{attribute 'qualified_only'}
{attribute 'to_string'}
TYPE eSeverity :
(
	None						:= 0,
	Info						:= 1,
	Warning 					:= 2,
	NormalShutdown				:= 3,
	QuickShutdown				:= 4,
	EmergencyShutdown			:= 5 //ONLY CALL FROM SAFETY PROGRAM		
);
END_TYPE

(* stored: Version 1.1.0.1, ProductVersion 3.1.4026.18
   DUT eSeverity: Id {0a1b3bf9-9c88-4dfa-9693-ad35466c57a4} *)
